FUNCTION_BLOCK ABSTRACT FB_ShapeDecorator IMPLEMENTS I_Shape
VAR
	_iDecoratedShape: I_Shape;
END_VAR

METHOD FB_init : BOOL
VAR_INPUT
	bInitRetains : BOOL; // if TRUE, the retain variables are initialized (warm start / cold start)
	bInCopyCode : BOOL;  // if TRUE, the instance afterwards gets moved into the copy code (online change)
	iDecoratedShape : I_Shape;
END_VAR
_iDecoratedShape := iDecoratedShape;
END_METHOD


METHOD ABSTRACT M_Draw : BOOL
END_METHOD

END_FUNCTION_BLOCK

(* stored: Version 1.1.0.1, ProductVersion 3.1.4024.12
   POU FB_ShapeDecorator: Id {b50439ab-ead7-48f7-9067-265d8e430227}, SpecialFunc None
   Method FB_init: Id {3510c160-9da0-4a5d-bae0-cc766fedd0c5}
   Method M_Draw: Id {500aee08-9f31-4a62-a84c-2b5663385250} *)
